FUNCTION_BLOCK CylControl
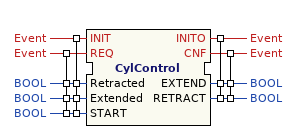
  EVENT_INPUT
    INIT WITH Retracted, Extended, START;
    REQ WITH Retracted, Extended, START;
  END_EVENT
  EVENT_OUTPUT
    INITO WITH EXTEND, RETRACT;
    CNF WITH EXTEND, RETRACT;
  END_EVENT
  VAR_INPUT
    Retracted : BOOL;
    Extended : BOOL;
    START : BOOL;
  END_VAR
  VAR_OUTPUT
    EXTEND : BOOL;
    RETRACT : BOOL;
  END_VAR
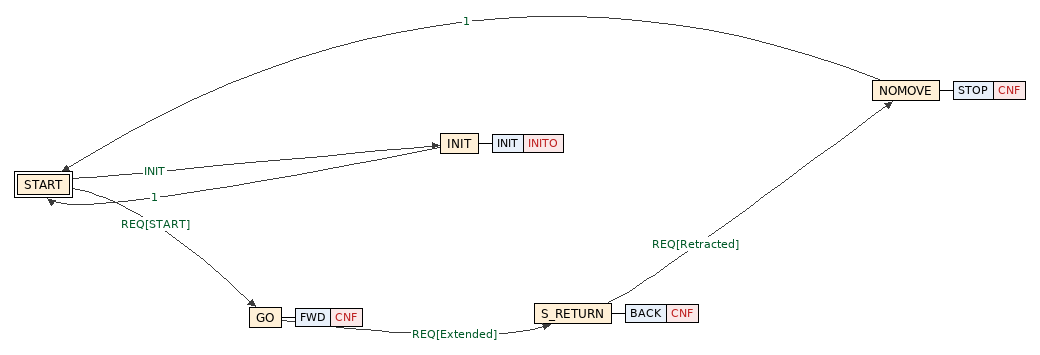
  EC_STATES
    START;
    INIT : INIT -> INITO;
    GO : FWD -> CNF;
    S_RETURN : BACK -> CNF;
    NOMOVE : STOP -> CNF;
  END_STATES
  EC_TRANSITIONS
    START TO INIT := INIT;
    INIT TO START := 1;
    START TO GO := REQ[START];
    GO TO S_RETURN := REQ[Extended];
    S_RETURN TO NOMOVE := REQ[Retracted];
    NOMOVE TO START := 1;
  END_TRANSITIONS
  ALGORITHM INIT IN ST:
EXTEND := FALSE;&#38;#10;RETRACT := FALSE;&#38;#10;
  END_ALGORITHM
  ALGORITHM REQ IN ST:

  END_ALGORITHM
  ALGORITHM FWD IN ST:
EXTEND := TRUE;&#38;#10;RETRACT := FALSE;&#38;#10;
  END_ALGORITHM
  ALGORITHM BACK IN ST:
EXTEND := FALSE;&#38;#10;RETRACT := TRUE;&#38;#10;
  END_ALGORITHM
  ALGORITHM STOP IN ST:
EXTEND := FALSE;&#38;#10;RETRACT := FALSE;&#38;#10;
  END_ALGORITHM
END_FUNCTION_BLOCK
